// TIA Portal project "4063_PLC" (V16)

(* hardware
DEVICE "S71500/ET200MP station_1"  S7-1500 station
   slot 0: "Telaio di montaggio_0"  Rack  6ES7 590-1***0-0AA0
   slot 1: "PLC_4063"  CPU 1511-1 PN  6ES7 511-1AK02-0AB0  V2.8
      slot 3: "Display CPU_1"  6ES7591-1AA00-0AA0
      slot 32768: "Interfaccia PROFINET_1"  X1
         slot 32769: "Porta_1"  X1 P1
         slot 32770: "Porta_2"  X1 P2
      slot 34817: "Virtual CP interface port_1"  Virtual CP interface port  Virtual CP interface port
   slot 2: "DI 16x24VDC HF_1"  DI 16x24VDC HF  6ES7 521-1BH00-0AB0  V2.2
   slot 3: "DQ 16x24VDC/0.5A HF_1"  DQ 16x24VDC/0.5A HF  6ES7 522-1BH01-0AB0  V1.1
   slot 4: "AQ 4xU/I ST_1"  AQ 4xU/I ST  6ES7 532-5HD00-0AB0  V2.2
   slot 5: "DI 16x24VDC HF_2"  DI 16x24VDC HF  6ES7 521-1BH00-0AB0  V2.2
   slot 6: "AQ 2xU/I ST_1"  AQ 2xU/I ST  6ES7 532-5NB00-0AB0  V1.0
   slot 7: "DQ 16x24VDC/0.5A HF_2"  DQ 16x24VDC/0.5A HF  6ES7 522-1BH01-0AB0  V1.1
   slot 8: "DI 16x24VDC HF_3"  DI 16x24VDC HF  6ES7 521-1BH00-0AB0  V2.2
   slot 9: "CP 1542-5_1"  CP 1542-5  6GK7 542-5FX00-0XE0  V2.0
DEVICE "SERVO_11"  GSD.Device
   slot 0: "UR"  Rail
DEVICE "SERVO_1"  GSD.Device
   slot 0: "UR"  Rail
DEVICE "SERVO_2"  GSD.Device
   slot 0: "UR"  Rail
DEVICE "SERVO_3"  GSD.Device
   slot 0: "UR"  Rail
DEVICE "SERVO_4"  GSD.Device
   slot 0: "UR"  Rail
DEVICE "SERVO_5"  GSD.Device
   slot 0: "UR"  Rail
DEVICE "SERVO_6"  GSD.Device
   slot 0: "UR"  Rail
*)

// ===== PLC "PLC_4063"  CPU 1511-1 PN =====

// folder: DataTypes

DATA_BLOCK "Binary_Numbers"   // DB3
{ S7_Optimized_Access := 'TRUE' }
VERSION : 0.1
   VAR
      Bool_Single_Bit : Bool := true;   // Boolean with possible states True or False
      String_Of_Byte : Byte := 100;   // Un operando del tipo di dati BYTE è una sequenza di 8 bit
      String_Of_Word : Word := 200;   // Un operando del tipo di dati WORD è una sequenza di 16 bit
      String_Of_Dword : DWord := 300;   // Un operando del tipo di dati DWORD è una sequenza di 32 bit
      String_Of_Lword : LWord := 400;   // Un operando del tipo di dati LWORD è una sequenza di 64 bit
   END_VAR
BEGIN
END_DATA_BLOCK

DATA_BLOCK "Integer_Numbers"   // DB6
{ S7_Optimized_Access := 'TRUE' }
VERSION : 0.1
   VAR
      Sint_Value : SInt;   // Un operando del tipo di dati SINT (Short INT) ha una lunghezza di 8 bit con segno
      Int_Value : Int;   // Un operando del tipo di dati INT ha una lunghezza pari a 16 bit con segno
      Dint_Value : DInt;   // Un operando del tipo di dati DINT (Double INT) ha una lunghezza pari a 32 bit con segno
      Usint_Value : USInt;   // Un operando del tipo di dati USINT (Unsigned Short INT) ha una lunghezza pari a 8 bit e contiene valori numerici senza segno
      Uint_Value : UInt;   // Un operando del tipo di dati UINT (Unsigned INT) ha una lunghezza pari a 16 bit e contiene valori numerici senza segno.
      Udint_Value : UDInt;   // Un operando del tipo di dati UDINT (Unsigned Double INT) ha una lunghezza pari a 32 bit e contiene valori numerici senza segno.
      LInt_Value : LInt;   // Un operando del tipo di dati LINT (Long INT) ha una lunghezza pari a 64 bit con segno
      Ulint_Value : ULInt;   // Un operando del tipo di dati ULINT (Unsigned Long INT) ha una lunghezza pari a 64 bit e contiene valori numerici senza segno.
   END_VAR
BEGIN
END_DATA_BLOCK

DATA_BLOCK "Float_Numbers"   // DB8
{ S7_Optimized_Access := 'TRUE' }
VERSION : 0.1
   VAR
      Real_Number : Real := 90.599;   // Gli operandi del tipo di dati REAL hanno una lunghezza pari a 32 bit, 1 bit segno, 8 bit esponente , 23 bit Mantissa
      Lreal_Number : LReal := -100.651989;   // Gli operandi del tipo di dati LREAL hanno una lunghezza pari a 64 bit, 1 bit segno, 11 bit esponente , 52 bit Mantissa
   END_VAR
BEGIN
END_DATA_BLOCK

DATA_BLOCK "Timers_Types"   // DB9
{ S7_Optimized_Access := 'TRUE' }
VERSION : 0.1
   VAR
      S5time_Value : S5Time := S5T#100ms;   // Il tipo di dati S5TIME memorizza la durata in formato BCD. La durata è il prodotto di un valore temporale compreso in un campo da 0 a 999 per una base temporale
      Time_Value : Time;   // Il contenuto di un operando del tipo di dati TIME viene interpretato in millisecondi. La rappresentazione comprende le indicazioni di giorni (d), ore (h), minuti (m), secondi (s) e millisecondi (ms).
      Ltime_Value : LTime;   // Il contenuto di un operando del tipo di dati LTIME viene interpretato in nanosecondi. La rappresentazione comprende le indicazioni di giorni (d), ore (h), minuti (m), secondi (s) e millisecondi (ms), microsecondi (us) e nanosecondi (ns).
   END_VAR
BEGIN
END_DATA_BLOCK

DATA_BLOCK "Date_Time"   // DB10
{ S7_Optimized_Access := 'TRUE' }
VERSION : 0.1
   VAR
      Date_value : Date;   // Il tipo di dati DATE salva una data come numero intero senza segno. La rappresentazione contiene l'anno, il mese e il giorno.
      Time_Of_Day : Time_Of_Day;   // Il tipo di dati TOD (TIME_OF_DAY) occupa una doppia parola e salva, come numero intero senza segno, il numero dei millisecondi a partire dalla mezzanotte (ore: 0:00).
      Ltime_Of_Day : LTime_Of_Day;   // Il tipo di dati LTOD (LTIME_OF_DAY) occupa due doppie parole e salva, come numero intero senza segno, il numero di nanosecondi a partire dalla mezzanotte (ore: 0:00).
      Date_And_Time : Date_And_Time;   // Il tipo di dati DT (DATE_AND_TIME) salva le indicazioni relative a data e ora in formato BCD.
      Date_And_Ltime : LDT;   // Il tipo di dati LDT (DATE_AND_LTIME) salva le indicazioni in nanosecondi relative a data e ora ad iniziare da 01.01.1970 0:0.
      Complete_DTL : DTL;   // Un operando del tipo di dati DTL ha una lunghezza pari a 12 byte e salva indicazioni relative a data e ora in una struttura predefinita.
   END_VAR
BEGIN
END_DATA_BLOCK

DATA_BLOCK "String_Types"   // DB11
{ S7_Optimized_Access := 'TRUE' }
VERSION : 0.1
   VAR
      "CHAR" : Char;   // Una variabile del tipo di dati CHAR (Character) ha una lunghezza di 8 bit e occupa un BYTE di memoria.
      WCHAR : WChar;   // Una variabile del tipo di dati WCHAR (Wide Characters) ha una lunghezza di 16 bit e occupa due BYTE di memoria.
      "STRING" : String;   // Un operando del tipo di dati STRING salva più caratteri in una stringa che può comprenderne al massimo 254.
      WSTRING : WString;   // Un operando con tipo di dati WSTRING (Wide Character String) salva più caratteri Unicode con tipo di dati WCHAR in una stringa
   END_VAR
BEGIN
END_DATA_BLOCK

DATA_BLOCK "PLC_data_Types"   // DB12
{ S7_Optimized_Access := 'TRUE' }
VERSION : 0.1
BEGIN
END_DATA_BLOCK

DATA_BLOCK "Structures_Types"   // DB13
{ S7_Optimized_Access := 'TRUE' }
VERSION : 0.1
   VAR
      STRUCTURE : Struct   // Is the equivalent of an Object Type with only attributes
         ANY_DATA : Bool;
      END_STRUCT;
   END_VAR
BEGIN
END_DATA_BLOCK

DATA_BLOCK "Array_Types"   // DB14
{ S7_Optimized_Access := 'TRUE' }
VERSION : 0.1
   VAR
      First_Array : Array[0..10] of HW_IOSYSTEM;   // Can be of any equal type of data
   END_VAR
BEGIN
END_DATA_BLOCK

DATA_BLOCK "System_Data_Types"   // DB17
{ S7_Optimized_Access := 'TRUE' }
VERSION : 0.1
   VAR
      IEC_TIMER : IEC_TIMER;
      IEC_LTIMER : IEC_LTIMER;
      IEC_SCOUNTER : IEC_SCOUNTER;
      IEC_COUNTER : IEC_COUNTER;
      IEC_UCOUNTER : IEC_UCOUNTER;
      IEC_DCOUNTER : IEC_DCOUNTER;
      IEC_LCOUNTER : IEC_LCOUNTER;
      IEC_ULCOUNTER : IEC_ULCOUNTER;
      ERROR_STRUCT : ErrorStruct;
      CREF : CREF;
      NREF : NREF;
   END_VAR
BEGIN
END_DATA_BLOCK

DATA_BLOCK "Hardware_Data_Types"   // DB18
{ S7_Optimized_Access := 'TRUE' }
VERSION : 0.1
   VAR
      HW_ANY : Hw_Any;   // Identificazione di un qualsiasi componente hardware, ad es. di un'unità.
      HW_DEVICE : Hw_Device;   // Identificazione di uno slave DP/PROFINET IO Device
      EVENT_ANY : Event_Any;   // Serve ad indicare un evento qualsiasi
      OB_ANY : OB_Any;   // Consente di indicare un blocco organizzativo qualsiasi.
      CONN_ANY : Conn_Any;   // Consente di indicare un collegamento qualsiasi.
   END_VAR
BEGIN
END_DATA_BLOCK

// folder: GET_Values

DATA_BLOCK "GET_Array_Data"   // DB2
{ S7_Optimized_Access := 'TRUE' }
VERSION : 0.1
   VAR
      data_array : Array[0..5] of Int;
      result_data_array : Array[0..100] of Int;
   END_VAR
BEGIN
   data_array[0] := 99;
   data_array[1] := 5;
   data_array[2] := 1;
   data_array[3] := 1000;
   data_array[4] := 1;
END_DATA_BLOCK

// folder: GET_Values/Bool_Values

DATA_BLOCK "GET_Time_Values"   // DB1
{ S7_Optimized_Access := 'TRUE' }
VERSION : 0.1
   VAR
      Timer_Random_Numbers : Time := T#5s;
   END_VAR
BEGIN
END_DATA_BLOCK

DATA_BLOCK "GET_Bool_Values"   // DB5
{ S7_Optimized_Access := 'TRUE' }
VERSION : 0.1
   VAR
      status_trigger_random_numbers : Bool;
      Timer_End_Pulse : Bool;
   END_VAR
BEGIN
END_DATA_BLOCK

// folder: PUT_Values/Bool_Values

DATA_BLOCK "PUT_Bool_Values"   // DB4
{ S7_Optimized_Access := 'TRUE' }
VERSION : 0.1
   VAR
      start_counting : Bool;
   END_VAR
BEGIN
END_DATA_BLOCK

// folder: System blocks/Program resources

DATA_BLOCK "IEC_Timer_0_DB"   // DB7
{ S7_Optimized_Access := 'TRUE' }
AUTHOR : Simatic
FAMILY : IEC
NAME : IEC_TMR
VERSION : 1.0
// stored: InstanceOfName IEC_TIMER
"IEC_TIMER"
BEGIN
END_DATA_BLOCK

// folder: (top level)

FUNCTION "Random_Number" : Void   // FC1, SCL
{ S7_Optimized_Access := 'TRUE' }
VERSION : 0.1
   VAR_INPUT
      "array" : Int;   // desired array length
      multiplier : Int;   // a=multiplier
      increment : Int;   // b=increment
      modulus : Int;   // m=modulus
      seed : Int;   // seed
   END_VAR
   VAR_OUTPUT
      Random_Number_list : Array[0..100] of Int;
   END_VAR
   VAR_TEMP
      index : Int;
      x0 : Int;
      array_check : Int;
      internal_multiplier : Int;
      internal_modulus : Int;
      internal_increment : Int;
      new_result : Int;
   END_VAR
   VAR CONSTANT
      zero : Int;
   END_VAR
BEGIN
   // index Identifier while looping 
   #index := 0;

   #x0 := #seed;
   #array_check := #array;
   #internal_multiplier := #multiplier;
   #internal_modulus := #modulus;
   #internal_increment := #increment;

   // Se i numeri sono maggiori di zero e internal_modulus è maggiore a tutti quindi e possibile generare 
   // dei numeri random 

   IF #internal_modulus > #zero AND
       #internal_multiplier > #zero AND
       #internal_increment > #zero AND
       #x0 > #zero AND
       #x0 < #internal_modulus AND
       #internal_multiplier < #internal_modulus AND
       #internal_increment < #internal_modulus THEN
       // Create and append random nuber to an Array 
       WHILE #array_check > #index DO

           #x0 := #internal_multiplier * (#x0 + #internal_increment);

           #new_result := #x0 / #internal_multiplier;

           #index := #index + 1;

           #Random_Number_list[#index] := ABS(#new_result);


       END_WHILE;
   END_IF;

   RETURN;
END_FUNCTION

ORGANIZATION_BLOCK "Main"   // OB1, LAD, ProgramCycle
TITLE = "Main Program Sweep (Cycle)"
{ S7_Optimized_Access := 'TRUE' }
VERSION : 0.1
   VAR_INPUT
      Initial_Call : Bool;   // Initial call of this OB
      Remanence : Bool;   // =True, if remanent data are available
   END_VAR
   VAR_TEMP
      Random_Number : Array[0..100] of Int;
   END_VAR
   VAR_TEMP   // added for the SCL form of the ladder/FBD networks
      _w1 : Bool;
      _w2 : Bool;
   END_VAR
BEGIN

REGION Network 1
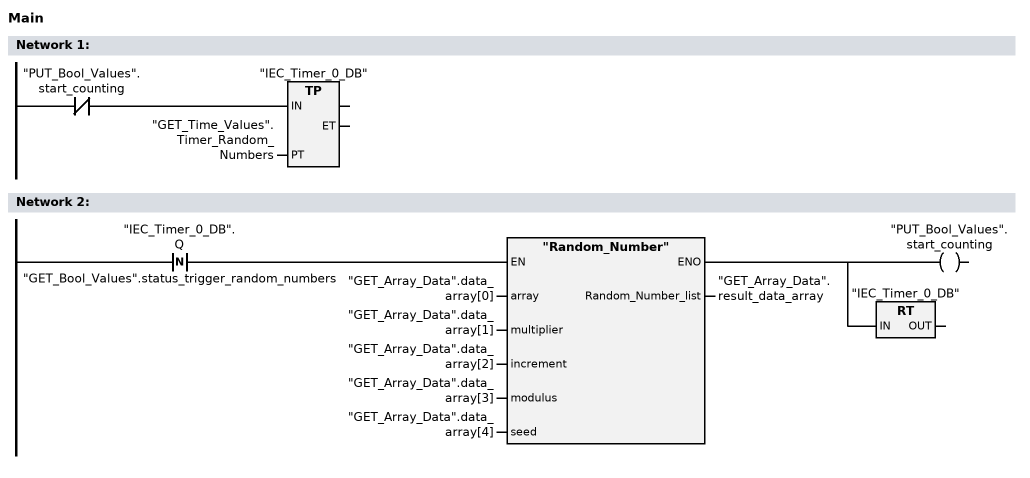
   "IEC_Timer_0_DB".TP(IN := NOT "PUT_Bool_Values".start_counting, PT := "GET_Time_Values".Timer_Random_Numbers);
END_REGION

REGION Network 2
   RUNG wire#powerrail
      N_Contact(operand := "IEC_Timer_0_DB".Q, bit := "GET_Bool_Values".status_trigger_random_numbers)
      "Random_Number"("array" := "GET_Array_Data".data_array[0], multiplier := "GET_Array_Data".data_array[1], increment := "GET_Array_Data".data_array[2], modulus := "GET_Array_Data".data_array[3], seed := "GET_Array_Data".data_array[4], Random_Number_list => "GET_Array_Data".result_data_array)
      wire#w1
      Coil( "PUT_Bool_Values".start_counting )
   END_RUNG
   RUNG wire#w1
      RT_Coil( "IEC_Timer_0_DB" )
   END_RUNG
   // the same network as SCL:
   #_w1 := NOT "IEC_Timer_0_DB".Q AND "GET_Bool_Values".status_trigger_random_numbers;   // falling edge of "IEC_Timer_0_DB".Q
   "GET_Bool_Values".status_trigger_random_numbers := "IEC_Timer_0_DB".Q;
   "Random_Number"(EN := #_w1,
                   "array" := "GET_Array_Data".data_array[0],
                   multiplier := "GET_Array_Data".data_array[1],
                   increment := "GET_Array_Data".data_array[2],
                   modulus := "GET_Array_Data".data_array[3],
                   seed := "GET_Array_Data".data_array[4],
                   Random_Number_list => "GET_Array_Data".result_data_array,
                   ENO => #_w2);
   "PUT_Bool_Values".start_counting := #_w2;
   IF #_w2 THEN RESET_TIMER("IEC_Timer_0_DB"); END_IF;
END_REGION

REGION Network 3 (SCL): Generate random numbers every (X) seconds
   IF "PUT_Bool_Values".start_counting THEN
       "GET_Array_Data".data_array[4] := "GET_Array_Data".result_data_array["GET_Array_Data".data_array[0]];
       "GET_Array_Data".data_array[3] := "GET_Array_Data".data_array[4] * 2;
   END_IF;
END_REGION

REGION Network 4 (SCL)
   "String_Types"."CHAR" := 'A';
   "String_Types"."STRING" := 'ABC';
   "String_Types"."WCHAR" := WCHAR#'a';
   "String_Types"."WSTRING" := WSTRING#'Hallo We... (La lunghezza attuale della stringa supera lo spazio disponibile sul display).';
END_REGION
END_ORGANIZATION_BLOCK